FUNCTION CheckDivLreal : LREAL
VAR_INPUT
	divisor		 		: LREAL;
END_VAR
VAR
END_VAR

IF divisor = 0 THEN
	CheckLrealZeroDiv_ErrCnt := CheckLrealZeroDiv_ErrCnt + 1;
	CheckDivLreal := 1;
ELSE
	CheckDivLreal := divisor;
END_IF

END_FUNCTION

(* stored: Version 1.1.0.1, ProductVersion 3.1.4024.9
   POU CheckDivLreal: Id {e35a8d6b-3b90-461f-887d-6ab3be1eaaa0}, SpecialFunc CheckDivReal64 *)
